// Mitsubishi GX Works2 project: Contador e temporizador   PLC: Q03UDV
// HelloWorld

PROGRAM MAIN
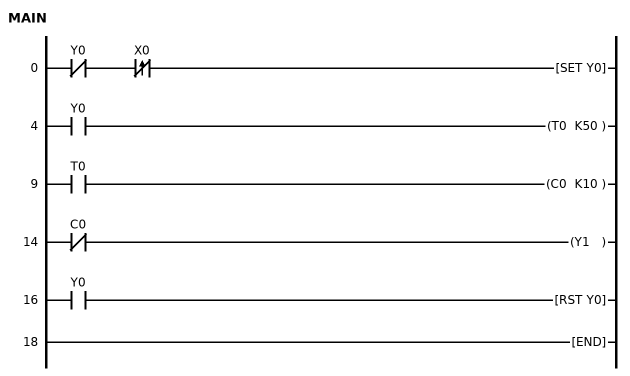
0     LDI     Y0
      ANDPI   X0
      SET     Y0
4     LD      Y0
      OUT     T0 K50
9     LD      T0
      OUT     C0 K10
14    LDI     C0
      OUT     Y1
16    LD      Y0
      RST     Y0
18    END
END_PROGRAM
